# EPICS substitutions: products/ITER/products/org.csstudio.iter.css.product/demo/m-TEST-BOY/src/main/epics/SharedTemplateApp/Db/rndm.substitutions
file rndm.db {
    pattern { IOC, COUNT, SCAN }
        { "A", "0", ".1 second" }
        { "A", "1", ".1 second" }
        { "A", "2", ".1 second" }
        { "A", "3", ".1 second" }
        { "A", "4", ".1 second" }
        { "A", "5", ".1 second" }
        { "A", "6", ".1 second" }
        { "A", "7", ".1 second" }
        { "A", "8", ".1 second" }
        { "A", "9", ".1 second" }
        { "A", "10", ".1 second" }
        { "A", "11", ".1 second" }
        { "A", "12", ".1 second" }
        { "A", "13", ".1 second" }
        { "A", "14", ".1 second" }
        { "A", "15", ".1 second" }
        { "A", "16", ".1 second" }
        { "A", "17", ".1 second" }
        { "A", "18", ".1 second" }
        { "A", "19", ".1 second" }
        { "A", "20", ".1 second" }
        { "A", "21", ".1 second" }
        { "A", "22", ".1 second" }
        { "A", "23", ".1 second" }
        { "A", "24", ".1 second" }
        { "A", "25", ".1 second" }
        { "A", "26", ".1 second" }
        { "A", "27", ".1 second" }
        { "A", "28", ".1 second" }
        { "A", "29", ".1 second" }
        { "A", "30", ".1 second" }
        { "A", "31", ".1 second" }
        { "A", "32", ".1 second" }
        { "A", "33", ".1 second" }
        { "A", "34", ".1 second" }
        { "A", "35", ".1 second" }
        { "A", "36", ".1 second" }
        { "A", "37", ".1 second" }
        { "A", "38", ".1 second" }
        { "A", "39", ".1 second" }
        { "A", "40", ".1 second" }
        { "A", "41", ".1 second" }
        { "A", "42", ".1 second" }
        { "A", "43", ".1 second" }
        { "A", "44", ".1 second" }
        { "A", "45", ".1 second" }
        { "A", "46", ".1 second" }
        { "A", "47", ".1 second" }
        { "A", "48", ".1 second" }
        { "A", "49", ".1 second" }
        { "A", "50", ".1 second" }
        { "A", "51", ".1 second" }
        { "A", "52", ".1 second" }
        { "A", "53", ".1 second" }
        { "A", "54", ".1 second" }
        { "A", "55", ".1 second" }
        { "A", "56", ".1 second" }
        { "A", "57", ".1 second" }
        { "A", "58", ".1 second" }
        { "A", "59", ".1 second" }
        { "A", "60", ".1 second" }
        { "A", "61", ".1 second" }
        { "A", "62", ".1 second" }
        { "A", "63", ".1 second" }
        { "A", "64", ".1 second" }
        { "A", "65", ".1 second" }
        { "A", "66", ".1 second" }
        { "A", "67", ".1 second" }
        { "A", "68", ".1 second" }
        { "A", "69", ".1 second" }
        { "A", "70", ".1 second" }
        { "A", "71", ".1 second" }
        { "A", "72", ".1 second" }
        { "A", "73", ".1 second" }
        { "A", "74", ".1 second" }
        { "A", "75", ".1 second" }
        { "A", "76", ".1 second" }
        { "A", "77", ".1 second" }
        { "A", "78", ".1 second" }
        { "A", "79", ".1 second" }
        { "A", "80", ".1 second" }
        { "A", "81", ".1 second" }
        { "A", "82", ".1 second" }
        { "A", "83", ".1 second" }
        { "A", "84", ".1 second" }
        { "A", "85", ".1 second" }
        { "A", "86", ".1 second" }
        { "A", "87", ".1 second" }
        { "A", "88", ".1 second" }
        { "A", "89", ".1 second" }
        { "A", "90", ".1 second" }
        { "A", "91", ".1 second" }
        { "A", "92", ".1 second" }
        { "A", "93", ".1 second" }
        { "A", "94", ".1 second" }
        { "A", "95", ".1 second" }
        { "A", "96", ".1 second" }
        { "A", "97", ".1 second" }
        { "A", "98", ".1 second" }
        { "A", "99", ".1 second" }
        { "A", "100", ".1 second" }
        { "A", "101", ".1 second" }
        { "A", "102", ".1 second" }
        { "A", "103", ".1 second" }
        { "A", "104", ".1 second" }
        { "A", "105", ".1 second" }
        { "A", "106", ".1 second" }
        { "A", "107", ".1 second" }
        { "A", "108", ".1 second" }
        { "A", "109", ".1 second" }
        { "A", "110", ".1 second" }
        { "A", "111", ".1 second" }
        { "A", "112", ".1 second" }
        { "A", "113", ".1 second" }
        { "A", "114", ".1 second" }
        { "A", "115", ".1 second" }
        { "A", "116", ".1 second" }
        { "A", "117", ".1 second" }
        { "A", "118", ".1 second" }
        { "A", "119", ".1 second" }
        { "A", "120", ".1 second" }
        { "A", "121", ".1 second" }
        { "A", "122", ".1 second" }
        { "A", "123", ".1 second" }
        { "A", "124", ".1 second" }
        { "A", "125", ".1 second" }
        { "A", "126", ".1 second" }
        { "A", "127", ".1 second" }
        { "A", "128", ".1 second" }
        { "A", "129", ".1 second" }
        { "A", "130", ".1 second" }
        { "A", "131", ".1 second" }
        { "A", "132", ".1 second" }
        { "A", "133", ".1 second" }
        { "A", "134", ".1 second" }
        { "A", "135", ".1 second" }
        { "A", "136", ".1 second" }
        { "A", "137", ".1 second" }
        { "A", "138", ".1 second" }
        { "A", "139", ".1 second" }
        { "A", "140", ".1 second" }
        { "A", "141", ".1 second" }
        { "A", "142", ".1 second" }
        { "A", "143", ".1 second" }
        { "A", "144", ".1 second" }
        { "A", "145", ".1 second" }
        { "A", "146", ".1 second" }
        { "A", "147", ".1 second" }
        { "A", "148", ".1 second" }
        { "A", "149", ".1 second" }
        { "A", "150", ".1 second" }
        { "A", "151", ".1 second" }
        { "A", "152", ".1 second" }
        { "A", "153", ".1 second" }
        { "A", "154", ".1 second" }
        { "A", "155", ".1 second" }
        { "A", "156", ".1 second" }
        { "A", "157", ".1 second" }
        { "A", "158", ".1 second" }
        { "A", "159", ".1 second" }
        { "A", "160", ".1 second" }
        { "A", "161", ".1 second" }
        { "A", "162", ".1 second" }
        { "A", "163", ".1 second" }
        { "A", "164", ".1 second" }
        { "A", "165", ".1 second" }
        { "A", "166", ".1 second" }
        { "A", "167", ".1 second" }
        { "A", "168", ".1 second" }
        { "A", "169", ".1 second" }
        { "A", "170", ".1 second" }
        { "A", "171", ".1 second" }
        { "A", "172", ".1 second" }
        { "A", "173", ".1 second" }
        { "A", "174", ".1 second" }
        { "A", "175", ".1 second" }
        { "A", "176", ".1 second" }
        { "A", "177", ".1 second" }
        { "A", "178", ".1 second" }
        { "A", "179", ".1 second" }
        { "A", "180", ".1 second" }
        { "A", "181", ".1 second" }
        { "A", "182", ".1 second" }
        { "A", "183", ".1 second" }
        { "A", "184", ".1 second" }
        { "A", "185", ".1 second" }
        { "A", "186", ".1 second" }
        { "A", "187", ".1 second" }
        { "A", "188", ".1 second" }
        { "A", "189", ".1 second" }
        { "A", "190", ".1 second" }
        { "A", "191", ".1 second" }
        { "A", "192", ".1 second" }
        { "A", "193", ".1 second" }
        { "A", "194", ".1 second" }
        { "A", "195", ".1 second" }
        { "A", "196", ".1 second" }
        { "A", "197", ".1 second" }
        { "A", "198", ".1 second" }
        { "A", "199", ".1 second" }
        { "A", "200", ".1 second" }
        { "A", "201", ".1 second" }
        { "A", "202", ".1 second" }
        { "A", "203", ".1 second" }
        { "A", "204", ".1 second" }
        { "A", "205", ".1 second" }
        { "A", "206", ".1 second" }
        { "A", "207", ".1 second" }
        { "A", "208", ".1 second" }
        { "A", "209", ".1 second" }
        { "A", "210", ".1 second" }
        { "A", "211", ".1 second" }
        { "A", "212", ".1 second" }
        { "A", "213", ".1 second" }
        { "A", "214", ".1 second" }
        { "A", "215", ".1 second" }
        { "A", "216", ".1 second" }
        { "A", "217", ".1 second" }
        { "A", "218", ".1 second" }
        { "A", "219", ".1 second" }
        { "A", "220", ".1 second" }
        { "A", "221", ".1 second" }
        { "A", "222", ".1 second" }
        { "A", "223", ".1 second" }
        { "A", "224", ".1 second" }
        { "A", "225", ".1 second" }
        { "A", "226", ".1 second" }
        { "A", "227", ".1 second" }
        { "A", "228", ".1 second" }
        { "A", "229", ".1 second" }
        { "A", "230", ".1 second" }
        { "A", "231", ".1 second" }
        { "A", "232", ".1 second" }
        { "A", "233", ".1 second" }
        { "A", "234", ".1 second" }
        { "A", "235", ".1 second" }
        { "A", "236", ".1 second" }
        { "A", "237", ".1 second" }
        { "A", "238", ".1 second" }
        { "A", "239", ".1 second" }
        { "A", "240", ".1 second" }
        { "A", "241", ".1 second" }
        { "A", "242", ".1 second" }
        { "A", "243", ".1 second" }
        { "A", "244", ".1 second" }
        { "A", "245", ".1 second" }
        { "A", "246", ".1 second" }
        { "A", "247", ".1 second" }
        { "A", "248", ".1 second" }
        { "A", "249", ".1 second" }
        { "A", "250", ".1 second" }
        { "A", "251", ".1 second" }
        { "A", "252", ".1 second" }
        { "A", "253", ".1 second" }
        { "A", "254", ".1 second" }
        { "A", "255", ".1 second" }
        { "A", "256", ".1 second" }
        { "A", "257", ".1 second" }
        { "A", "258", ".1 second" }
        { "A", "259", ".1 second" }
        { "A", "260", ".1 second" }
        { "A", "261", ".1 second" }
        { "A", "262", ".1 second" }
        { "A", "263", ".1 second" }
        { "A", "264", ".1 second" }
        { "A", "265", ".1 second" }
        { "A", "266", ".1 second" }
        { "A", "267", ".1 second" }
        { "A", "268", ".1 second" }
        { "A", "269", ".1 second" }
        { "A", "270", ".1 second" }
        { "A", "271", ".1 second" }
        { "A", "272", ".1 second" }
        { "A", "273", ".1 second" }
        { "A", "274", ".1 second" }
        { "A", "275", ".1 second" }
        { "A", "276", ".1 second" }
        { "A", "277", ".1 second" }
        { "A", "278", ".1 second" }
        { "A", "279", ".1 second" }
        { "A", "280", ".1 second" }
        { "A", "281", ".1 second" }
        { "A", "282", ".1 second" }
        { "A", "283", ".1 second" }
        { "A", "284", ".1 second" }
        { "A", "285", ".1 second" }
        { "A", "286", ".1 second" }
        { "A", "287", ".1 second" }
        { "A", "288", ".1 second" }
        { "A", "289", ".1 second" }
        { "A", "290", ".1 second" }
        { "A", "291", ".1 second" }
        { "A", "292", ".1 second" }
        { "A", "293", ".1 second" }
        { "A", "294", ".1 second" }
        { "A", "295", ".1 second" }
        { "A", "296", ".1 second" }
        { "A", "297", ".1 second" }
        { "A", "298", ".1 second" }
        { "A", "299", ".1 second" }
        { "A", "300", ".1 second" }
        { "A", "301", ".1 second" }
        { "A", "302", ".1 second" }
        { "A", "303", ".1 second" }
        { "A", "304", ".1 second" }
        { "A", "305", ".1 second" }
        { "A", "306", ".1 second" }
        { "A", "307", ".1 second" }
        { "A", "308", ".1 second" }
        { "A", "309", ".1 second" }
        { "A", "310", ".1 second" }
        { "A", "311", ".1 second" }
        { "A", "312", ".1 second" }
        { "A", "313", ".1 second" }
        { "A", "314", ".1 second" }
        { "A", "315", ".1 second" }
        { "A", "316", ".1 second" }
        { "A", "317", ".1 second" }
        { "A", "318", ".1 second" }
        { "A", "319", ".1 second" }
        { "A", "320", ".1 second" }
        { "A", "321", ".1 second" }
        { "A", "322", ".1 second" }
        { "A", "323", ".1 second" }
        { "A", "324", ".1 second" }
        { "A", "325", ".1 second" }
        { "A", "326", ".1 second" }
        { "A", "327", ".1 second" }
        { "A", "328", ".1 second" }
        { "A", "329", ".1 second" }
        { "A", "330", ".1 second" }
        { "A", "331", ".1 second" }
        { "A", "332", ".1 second" }
        { "A", "333", ".1 second" }
        { "A", "334", ".1 second" }
        { "A", "335", ".1 second" }
        { "A", "336", ".1 second" }
        { "A", "337", ".1 second" }
        { "A", "338", ".1 second" }
        { "A", "339", ".1 second" }
        { "A", "340", ".1 second" }
        { "A", "341", ".1 second" }
        { "A", "342", ".1 second" }
        { "A", "343", ".1 second" }
        { "A", "344", ".1 second" }
        { "A", "345", ".1 second" }
        { "A", "346", ".1 second" }
        { "A", "347", ".1 second" }
        { "A", "348", ".1 second" }
        { "A", "349", ".1 second" }
        { "A", "350", ".1 second" }
        { "A", "351", ".1 second" }
        { "A", "352", ".1 second" }
        { "A", "353", ".1 second" }
        { "A", "354", ".1 second" }
        { "A", "355", ".1 second" }
        { "A", "356", ".1 second" }
        { "A", "357", ".1 second" }
        { "A", "358", ".1 second" }
        { "A", "359", ".1 second" }
        { "A", "360", ".1 second" }
        { "A", "361", ".1 second" }
        { "A", "362", ".1 second" }
        { "A", "363", ".1 second" }
        { "A", "364", ".1 second" }
        { "A", "365", ".1 second" }
        { "A", "366", ".1 second" }
        { "A", "367", ".1 second" }
        { "A", "368", ".1 second" }
        { "A", "369", ".1 second" }
        { "A", "370", ".1 second" }
        { "A", "371", ".1 second" }
        { "A", "372", ".1 second" }
        { "A", "373", ".1 second" }
        { "A", "374", ".1 second" }
        { "A", "375", ".1 second" }
        { "A", "376", ".1 second" }
        { "A", "377", ".1 second" }
        { "A", "378", ".1 second" }
        { "A", "379", ".1 second" }
        { "A", "380", ".1 second" }
        { "A", "381", ".1 second" }
        { "A", "382", ".1 second" }
        { "A", "383", ".1 second" }
        { "A", "384", ".1 second" }
        { "A", "385", ".1 second" }
        { "A", "386", ".1 second" }
        { "A", "387", ".1 second" }
        { "A", "388", ".1 second" }
        { "A", "389", ".1 second" }
        { "A", "390", ".1 second" }
        { "A", "391", ".1 second" }
        { "A", "392", ".1 second" }
        { "A", "393", ".1 second" }
        { "A", "394", ".1 second" }
        { "A", "395", ".1 second" }
        { "A", "396", ".1 second" }
        { "A", "397", ".1 second" }
        { "A", "398", ".1 second" }
        { "A", "399", ".1 second" }
        { "A", "400", ".1 second" }
        { "A", "401", ".1 second" }
        { "A", "402", ".1 second" }
        { "A", "403", ".1 second" }
        { "A", "404", ".1 second" }
        { "A", "405", ".1 second" }
        { "A", "406", ".1 second" }
        { "A", "407", ".1 second" }
        { "A", "408", ".1 second" }
        { "A", "409", ".1 second" }
        { "A", "410", ".1 second" }
        { "A", "411", ".1 second" }
        { "A", "412", ".1 second" }
        { "A", "413", ".1 second" }
        { "A", "414", ".1 second" }
        { "A", "415", ".1 second" }
        { "A", "416", ".1 second" }
        { "A", "417", ".1 second" }
        { "A", "418", ".1 second" }
        { "A", "419", ".1 second" }
        { "A", "420", ".1 second" }
        { "A", "421", ".1 second" }
        { "A", "422", ".1 second" }
        { "A", "423", ".1 second" }
        { "A", "424", ".1 second" }
        { "A", "425", ".1 second" }
        { "A", "426", ".1 second" }
        { "A", "427", ".1 second" }
        { "A", "428", ".1 second" }
        { "A", "429", ".1 second" }
        { "A", "430", ".1 second" }
        { "A", "431", ".1 second" }
        { "A", "432", ".1 second" }
        { "A", "433", ".1 second" }
        { "A", "434", ".1 second" }
        { "A", "435", ".1 second" }
        { "A", "436", ".1 second" }
        { "A", "437", ".1 second" }
        { "A", "438", ".1 second" }
        { "A", "439", ".1 second" }
        { "A", "440", ".1 second" }
        { "A", "441", ".1 second" }
        { "A", "442", ".1 second" }
        { "A", "443", ".1 second" }
        { "A", "444", ".1 second" }
        { "A", "445", ".1 second" }
        { "A", "446", ".1 second" }
        { "A", "447", ".1 second" }
        { "A", "448", ".1 second" }
        { "A", "449", ".1 second" }
        { "A", "450", ".1 second" }
        { "A", "451", ".1 second" }
        { "A", "452", ".1 second" }
        { "A", "453", ".1 second" }
        { "A", "454", ".1 second" }
        { "A", "455", ".1 second" }
        { "A", "456", ".1 second" }
        { "A", "457", ".1 second" }
        { "A", "458", ".1 second" }
        { "A", "459", ".1 second" }
        { "A", "460", ".1 second" }
        { "A", "461", ".1 second" }
        { "A", "462", ".1 second" }
        { "A", "463", ".1 second" }
        { "A", "464", ".1 second" }
        { "A", "465", ".1 second" }
        { "A", "466", ".1 second" }
        { "A", "467", ".1 second" }
        { "A", "468", ".1 second" }
        { "A", "469", ".1 second" }
        { "A", "470", ".1 second" }
        { "A", "471", ".1 second" }
        { "A", "472", ".1 second" }
        { "A", "473", ".1 second" }
        { "A", "474", ".1 second" }
        { "A", "475", ".1 second" }
        { "A", "476", ".1 second" }
        { "A", "477", ".1 second" }
        { "A", "478", ".1 second" }
        { "A", "479", ".1 second" }
        { "A", "480", ".1 second" }
        { "A", "481", ".1 second" }
        { "A", "482", ".1 second" }
        { "A", "483", ".1 second" }
        { "A", "484", ".1 second" }
        { "A", "485", ".1 second" }
        { "A", "486", ".1 second" }
        { "A", "487", ".1 second" }
        { "A", "488", ".1 second" }
        { "A", "489", ".1 second" }
        { "A", "490", ".1 second" }
        { "A", "491", ".1 second" }
        { "A", "492", ".1 second" }
        { "A", "493", ".1 second" }
        { "A", "494", ".1 second" }
        { "A", "495", ".1 second" }
        { "A", "496", ".1 second" }
        { "A", "497", ".1 second" }
        { "A", "498", ".1 second" }
        { "A", "499", ".1 second" }
        { "A", "500", ".1 second" }
        { "A", "501", ".1 second" }
        { "A", "502", ".1 second" }
        { "A", "503", ".1 second" }
        { "A", "504", ".1 second" }
        { "A", "505", ".1 second" }
        { "A", "506", ".1 second" }
        { "A", "507", ".1 second" }
        { "A", "508", ".1 second" }
        { "A", "509", ".1 second" }
        { "A", "510", ".1 second" }
        { "A", "511", ".1 second" }
        { "A", "512", ".1 second" }
        { "A", "513", ".1 second" }
        { "A", "514", ".1 second" }
        { "A", "515", ".1 second" }
        { "A", "516", ".1 second" }
        { "A", "517", ".1 second" }
        { "A", "518", ".1 second" }
        { "A", "519", ".1 second" }
}
